(* IEC 61131-3 sources: SJ_AGV/PLC/Vehicle_specfic_functions, 3 files *)

(* ---- BMS_CHG_FB.ST ---- *)
FUNCTION_BLOCK BMS_CHG_FB
VAR_EXTERNAL

END_VAR

VAR_INPUT

END_VAR

VAR_OUTPUT

END_VAR

VAR
	StepDelay : TON;
	ManualStepDelay : TON;
	CheckChargeDoneStepDelay : TON;

	 ChageTimer : TON;
	 ChargeFullFlag : BOOL;

	 AutoChargeStep : INT := 0;
	 ChargePnt : DINT := 0;

	 FastChargeFlag : BOOL;
	 FastChargeTimer : TON;
	 FastChargeTimeOver : BOOL;

END_VAR
(* Check Manual Charge *)

if PLC_RX03_Bit_ChrgReqL_A = TRUE and PLC_TX01_Bit_ManMode = TRUE and PLC_RX03_Bit_Charging_L = FALSE then
	NDC8.SDIO.DigitalOutput16_Charger := TRUE;
	PLC_TX01_Bit_ChrgSelL_A := TRUE;
	StopCharge := TRUE;

	(* Full Charge Point check *)
	if NDC8.PointTrigger.Bit14_Full_Chrg = FALSE then
		PLC_TX01_Bit_TRChg_Pnt := TRUE;
	else
		PLC_TX01_Bit_TRChg_Pnt := FALSE;
	end_if;

	g_BattLim_NG := FALSE;
	INPUT.LowBattery := FALSE;
	NDC8.Userdefined.LowBatSim := FALSE;
	OM_PLC_W1_Bit_SetLowBatt := FALSE;

	ManualStepDelay(IN := TRUE, PT := t#1s);

	if ManualStepDelay.Q Then
		PLC_TX04_Bit_ChrgCmdL_A := TRUE;
		ManualStepDelay(IN := FALSE);
	end_if;

elsif PLC_RX03_Bit_ChrgReqR_A = TRUE and PLC_TX01_Bit_ManMode = TRUE and PLC_RX03_Bit_Charging_R = FALSE then
	NDC8.SDIO.DigitalOutput16_Charger := TRUE;
	PLC_TX01_Bit_ChrgSelR_A := TRUE;
	StopCharge := TRUE;

	(* Full Charge Point check *)
	if NDC8.PointTrigger.Bit14_Full_Chrg = FALSE then
		PLC_TX01_Bit_TRChg_Pnt := TRUE;
	else
		PLC_TX01_Bit_TRChg_Pnt := FALSE;
	end_if;

	g_BattLim_NG := FALSE;
	INPUT.LowBattery := FALSE;
	NDC8.Userdefined.LowBatSim := FALSE;
	OM_PLC_W1_Bit_SetLowBatt := FALSE;

	ManualStepDelay(IN := TRUE, PT := t#1s);

	if ManualStepDelay.Q Then
		PLC_TX04_Bit_ChrgCmdR_A := TRUE;
		ManualStepDelay(IN := FALSE);
	end_if;

elsif (PLC_RX03_Bit_ChrgReqL_A = FALSE and PLC_RX03_Bit_ChrgReqR_A = FALSE) and PLC_TX01_Bit_ManMode = TRUE then
	NDC8.SDIO.DigitalOutput16_Charger := FALSE;

	PLC_TX04_Bit_ChrgCmdL_A := FALSE;
	PLC_TX04_Bit_ChrgCmdR_A := FALSE;

	PLC_TX01_Bit_TRChg_Pnt := FALSE;

	ManualStepDelay(IN := TRUE, PT := t#1s);

	if ManualStepDelay.Q Then
		PLC_TX01_Bit_ChrgSelL_A := FALSE;
		PLC_TX01_Bit_ChrgSelR_A := FALSE;
		StopCharge := FALSE;
		ManualStepDelay(IN := FALSE);
		INPUT.LowBattery := FALSE;
	end_if;

end_if;

case AutoChargeStep of

	0:

		if (INPUT.Auto = TRUE and NDC8.Automatic.ExecDriveCommand = FALSE ) and
			((NDC8.PointTrigger.Bit9_Chrg_Right = TRUE and NDC8.PointTrigger.Bit10_Chrg_Left = FALSE) or (NDC8.PointTrigger.Bit9_Chrg_Right = FALSE and NDC8.PointTrigger.Bit10_Chrg_Left = TRUE)) and
			(PLC_RX01_Bit_ChrgEmg = FALSE) then
			AutoChargeStep := 70;
			g_ChargeDone := FALSE;
			ChargePnt := NDC8.LayoutPosition.Point;
		end_if;

		OM_PLC_Word9 := INT_TO_WORD(NDC8.OMPLC.Round_om);

		OM_PLC_W9_Bit_ChgP_Err := FALSE;

		NDC8.OMPLC.Round_om := WORD_TO_INT(OM_PLC_Word9);

(* Charge the battery Host Order *)
	70:

		if NDC8.PointTrigger.Bit9_Chrg_Right = TRUE and NDC8.PointTrigger.Bit10_Chrg_Left = FALSE then
			PLC_TX01_Bit_ChrgSelR_A := TRUE;
		elsif NDC8.PointTrigger.Bit9_Chrg_Right = FALSE and NDC8.PointTrigger.Bit10_Chrg_Left = TRUE then
			PLC_TX01_Bit_ChrgSelL_A := TRUE;
		end_if;

		(* Full Charge Point check *)
		if NDC8.PointTrigger.Bit14_Full_Chrg = FALSE then
			PLC_TX01_Bit_TRChg_Pnt := TRUE;
		else
			PLC_TX01_Bit_TRChg_Pnt := FALSE;
		end_if;

		OM_PLC_Word9 := INT_TO_WORD(NDC8.OMPLC.Round_om);

		PLC_TX01_Bit_Cancel_ST2 := not OM_PLC_W9_Bit_Enable_Err;
		OM_PLC_W9_Bit_ChgP_Err := FALSE;

		if NDC8.PLC_Application.TxStatusBit9_EStop = TRUE then
			AutoChargeStep := 999;
		elsif PLC_RX01_Bit_ChrgEmg = TRUE then
			AutoChargeStep := 999;
		elsif PLC_RX03_Bit_Round_ChgP = TRUE then
			OM_PLC_W9_Bit_ChgP_Err := TRUE;
			AutoChargeStep := 72;
		elsif PLC_RX01_Bit_ChrgBrk = TRUE then
			AutoChargeStep := 72;
		elsif INPUT.Auto = FALSE then
			AutoChargeStep := 72;
		end_if;

		NDC8.OMPLC.Round_om := WORD_TO_INT(OM_PLC_Word9);

		StopCharge := TRUE;

		(* Check Charge Idle*)
		if PLC_RX03_Bit_CP_HP = TRUE then
			StepDelay(IN:=TRUE, PT:=t#2s);
			if StepDelay.Q then
				StepDelay(IN:=FALSE);
				AutoChargeStep := 71;
			end_if;

		end_if;

	71:

		OM_PLC_Word9 := INT_TO_WORD(NDC8.OMPLC.Round_om);

		PLC_TX01_Bit_Cancel_ST2 := not OM_PLC_W9_Bit_Enable_Err;

		OM_PLC_W9_Bit_ChgP_Err := FALSE;

		if NDC8.PLC_Application.TxStatusBit9_EStop = TRUE then
			AutoChargeStep := 999;
		elsif PLC_RX01_Bit_ChrgEmg = TRUE then
			AutoChargeStep := 999;
		elsif PLC_RX03_Bit_Round_ChgP = TRUE then
			OM_PLC_W9_Bit_ChgP_Err := TRUE;
			AutoChargeStep := 72;
		elsif PLC_RX01_Bit_ChrgBrk = TRUE then
			AutoChargeStep := 72;
		elsif INPUT.Auto = FALSE then
			AutoChargeStep := 72;
		end_if;

		NDC8.OMPLC.Round_om := WORD_TO_INT(OM_PLC_Word9);

		PLC_TX04_Bit_ChrgCmdL_A := NDC8.PointTrigger.Bit10_Chrg_Left;
		PLC_TX04_Bit_ChrgCmdR_A := NDC8.PointTrigger.Bit9_Chrg_Right;

		NDC8.SDIO.DigitalOutput16_Charger := TRUE;

		OM_PLC_Word1 := INT_TO_WORD(NDC8.OMPLC.ChargeOM);
		OM_PLC_Word2 := INT_TO_WORD(NDC8.OMPLC.Stop_OM);

		g_BattLim_NG := FALSE;
		INPUT.LowBattery := FALSE;
		NDC8.Userdefined.LowBatSim := FALSE;
		OM_PLC_W1_Bit_SetLowBatt := FALSE;

		if NDC8.PointTrigger.Bit14_Full_Chrg = TRUE then
			if (g_ChargeDone or PLC_RX01_Bit_ChrgEmg) then
				AutoChargeStep := 72;
			end_if;
		else
			if (NDC8.Automatic.ExecDriveCommand = TRUE or PLC_RX01_Bit_ChrgEmg) or g_ChargeDone or FastChargeTimeOver then
				AutoChargeStep := 72;
			end_if;
		end_if;

	72:

		OM_PLC_Word9 := INT_TO_WORD(NDC8.OMPLC.Round_om);

		PLC_TX01_Bit_Cancel_ST2 := not OM_PLC_W9_Bit_Enable_Err;

		NDC8.OMPLC.Round_om := WORD_TO_INT(OM_PLC_Word9);

		if PLC_RX01_Bit_ChrgEmg = TRUE then
			AutoChargeStep := 999;
		end_if;

		if NDC8.PLC_Application.TxStatusBit9_EStop = TRUE then
			AutoChargeStep := 999;
		end_if;

		PLC_TX04_Bit_ChrgCmdL_A := FALSE;
		PLC_TX04_Bit_ChrgCmdR_A := FALSE;

		NDC8.SDIO.DigitalOutput16_Charger := FALSE;

		OM_PLC_Word1 := INT_TO_WORD(NDC8.OMPLC.ChargeOM);

		OM_PLC_W1_Bit_SetLowBatt := FALSE;

		NDC8.OMPLC.ChargeOM := WORD_TO_INT(OM_PLC_Word1);

		StepDelay(IN:=TRUE, PT:=t#5s);
		if StepDelay.Q then
			StepDelay(IN:=FALSE);
			AutoChargeStep := 73;
		end_if;

	73:

		PLC_TX01_Bit_ChrgSelL_A := FALSE;
		PLC_TX01_Bit_ChrgSelR_A := FALSE;

		OM_PLC_Word9 := INT_TO_WORD(NDC8.OMPLC.Round_om);

		PLC_TX01_Bit_Cancel_ST2 := not OM_PLC_W9_Bit_Enable_Err;

		NDC8.OMPLC.Round_om := WORD_TO_INT(OM_PLC_Word9);

		if PLC_RX01_Bit_ChrgEmg = TRUE then
			AutoChargeStep := 999;
		end_if;

		if NDC8.PLC_Application.TxStatusBit9_EStop = TRUE then
			AutoChargeStep := 999;
		end_if;

		if PLC_RX03_Bit_CP_HP then
			StepDelay(IN:=TRUE, PT:=t#1s);
			if StepDelay.Q then
				StepDelay(IN:=FALSE);
				StopCharge := FALSE;
				AutoChargeStep := 74;
			end_if;
		end_if;

	74:

		OM_PLC_Word9 := INT_TO_WORD(NDC8.OMPLC.Round_om);

		PLC_TX01_Bit_Cancel_ST2 := not OM_PLC_W9_Bit_Enable_Err;

		NDC8.OMPLC.Round_om := WORD_TO_INT(OM_PLC_Word9);

		if PLC_RX01_Bit_ChrgEmg = TRUE then
			AutoChargeStep := 999;
		end_if;

		if NDC8.PLC_Application.TxStatusBit9_EStop = TRUE then
			AutoChargeStep := 999;
		end_if;

		if INPUT.Auto = FALSE then
			AutoChargeStep := 0;
		end_if;

		if NDC8.LayoutPosition.Point <> ChargePnt or NDC8.PLC_Application.TxStatusBit4_LowBatt = TRUE then
			AutoChargeStep := 0;
		end_if;

	999:
		PLC_TX04_Bit_ChrgCmdL_A := FALSE;
		PLC_TX04_Bit_ChrgCmdR_A := FALSE;

		PLC_TX01_Bit_TRChg_Pnt := FALSE;

		StepDelay(IN:=TRUE, PT:=t#1s);
		if StepDelay.Q then
			StepDelay(IN:=FALSE);
			PLC_TX01_Bit_ChrgSelL_A := FALSE;
			PLC_TX01_Bit_ChrgSelR_A := FALSE;
			AutoChargeStep := 0;
			INPUT.LowBattery := FALSE;
		end_if;

		NDC8.SDIO.DigitalOutput16_Charger := FALSE;

		OM_PLC_Word1 := INT_TO_WORD(NDC8.OMPLC.ChargeOM);

		OM_PLC_W1_Bit_SetLowBatt := FALSE;

		NDC8.OMPLC.ChargeOM := WORD_TO_INT(OM_PLC_Word1);

		StopCharge := FALSE;

end_case;

(* Charge Complete Check *)
if (NDC8.PointTrigger.Bit9_Chrg_Right = TRUE or NDC8.PointTrigger.Bit10_Chrg_Left = TRUE) or PLC_TX01_Bit_ManMode = TRUE then
	if(NDC8.CAN_IO_3.DigitalInput5_BatTmp25_i = TRUE and
		NDC8.CAN_IO_3.DigitalInput6_BatTmp40_i = TRUE and
		NDC8.CAN_IO_3.DigitalInput7_BatTmp55_i = TRUE and
		g_BatteryVoltage >= NDC8.UserDefined.Integer32_40_ChgComV1) then
		g_ChargeDone := TRUE;
		g_ChargeTempErr := FALSE;
	elsif (NDC8.CAN_IO_3.DigitalInput5_BatTmp25_i = FALSE and
		NDC8.CAN_IO_3.DigitalInput6_BatTmp40_i = TRUE and
		NDC8.CAN_IO_3.DigitalInput7_BatTmp55_i = TRUE and
		g_BatteryVoltage >= NDC8.UserDefined.Integer32_41_ChgComV2) then
		g_ChargeDone := TRUE;
		g_ChargeTempErr := FALSE;
	elsif (NDC8.CAN_IO_3.DigitalInput5_BatTmp25_i = FALSE and
		NDC8.CAN_IO_3.DigitalInput6_BatTmp40_i = FALSE and
		NDC8.CAN_IO_3.DigitalInput7_BatTmp55_i = TRUE and
		g_BatteryVoltage >= NDC8.UserDefined.Integer32_42_ChgComV3) then
		g_ChargeDone := TRUE;
		g_ChargeTempErr := FALSE;
	elsif (NDC8.CAN_IO_3.DigitalInput5_BatTmp25_i = FALSE and
		NDC8.CAN_IO_3.DigitalInput6_BatTmp40_i = FALSE and
		NDC8.CAN_IO_3.DigitalInput7_BatTmp55_i = FALSE) then
		g_ChargeDone := FALSE;
		g_ChargeTempErr := TRUE;
	else
		g_ChargeDone := FALSE;
		g_ChargeTempErr := FALSE;
	end_if;

elsif (NDC8.CAN_IO_3.DigitalInput5_BatTmp25_i = FALSE and
		NDC8.CAN_IO_3.DigitalInput6_BatTmp40_i = FALSE and
		NDC8.CAN_IO_3.DigitalInput7_BatTmp55_i = FALSE) then

	g_ChargeDone := FALSE;
	g_ChargeTempErr := TRUE;
else
	g_ChargeDone := FALSE;
	g_ChargeTempErr := FALSE;
end_if;

(* Charge Over Time Check *)

	ChargeFullFlag  := NDC8.SDIO.DigitalOutput16_Charger = TRUE and NDC8.PointTrigger.Bit14_Full_Chrg = TRUE;

	ChageTimer(IN:= ChargeFullFlag, PT:=t#1800s);

	if ChageTimer.Q then
		g_ChargeOverTime := TRUE;
	end_if;

	if ChargeFullFlag = FALSE then
		g_ChargeOverTime := FALSE;
	end_if;

(* Fast Charge Time Check *)

	FastChargeFlag := NDC8.SDIO.DigitalOutput16_Charger = TRUE and NDC8.PointTrigger.Bit14_Full_Chrg = FALSE;

	FastChargeTimer(IN:= FastChargeFlag, PT:=t#600s);

	if FastChargeTimer.Q then
		FastChargeTimeOver := TRUE;
	end_if;

	if FastChargeFlag = FALSE then
		FastChargeTimeOver := FALSE;
	end_if;

(* Check BMS Error Status *)
if NDC8.SDIO.DigitalInput2_BTN_RST = FALSE and
	(PLC_RX01_Bit_ChrgEmg = TRUE
	or g_ChargeDone = TRUE
	or g_ChargeOverTime = TRUE
	or g_ChargeTempErr = TRUE) then

		PLC_TX04_Bit_ChrgCmdL_A := FALSE;
		PLC_TX04_Bit_ChrgCmdR_A := FALSE;

		NDC8.SDIO.DigitalOutput16_Charger := FALSE;

		CheckChargeDoneStepDelay(IN := TRUE, PT := t#1s);

		if CheckChargeDoneStepDelay.Q then
			CheckChargeDoneStepDelay(IN := FALSE);
			PLC_TX01_Bit_ChrgSelL_A := FALSE;
			PLC_TX01_Bit_ChrgSelR_A := FALSE;
		end_if;

end_if;

(* Let Vehicle Stop *)
(*
if PLC_TX04_Bit_ChrgCmdL_A = TRUE or PLC_TX04_Bit_ChrgCmdR_A = TRUE or
	PLC_RX03_Bit_CP_HP = FALSE or
	AutoChargeStep = 70 or AutoChargeStep = 71 or AutoChargeStep = 72 or AutoChargeStep = 73 then
	StopCharge := TRUE;
end_if;
*)

END_FUNCTION_BLOCK

(* ---- MITSUBISHIMODBUS_FB.ST ---- *)
FUNCTION_BLOCK MITSUBISHIMODBUS_FB
VAR_EXTERNAL

	ConvWord:WORD;			(*Sum of the two first bytes*)

	ConvByteL:Byte;			(*Low byte*)
	ConvByteH:Byte;			(*High byte*)
END_VAR

VAR_INPUT
	ComStart : bool := TRUE;
END_VAR

VAR_OUTPUT

END_VAR

VAR
	BMS_BatLowSel : INT;
	BMS_BatLow : BOOL;

	TP_PB_NoSelTimer : TON;

	Debug_PB_Cont : BOOL := FALSE;
	Debug_PB_Finish : BOOL := FALSE;
	Debug_PB_Cancel : BOOL := FALSE;
	Debug_PB_Change : BOOL := FALSE;

	RST_Flag : BOOL;
	RST_R : R_Trig;

	RST_Keep : BOOL;
	RST_Keep_Timer : TON;

	BatLow : BOOL;

	TempInt : int;
	TempWord : word;
	WordL :int;
	WordH :int;

	FinalPnt : DINT;

	SwitchHostFlag : BOOL;
	Host_R : R_Trig;
	Host_R_Flag : BOOL;

	Host_R_Delay : TON;

	init  : bool := false;
	ComStep : int := 0;

	serial_read : NDC8_SERIAL_READ;
	serial_write : NDC8_SERIAL_WRITE;

	to_bytes 		: NDC8_STRING_TO_BYTES;
	to_string		: NDC8_BYTES_TO_STRING;

	PLC_LastHeartBeat : BOOL;
	PLC_HeartBeatNoChange : BOOL;

	PLC_HeartBeatTimeout : TON;

	LoadDataSendFlag : BOOL;
	UnloadDataSendFlag : BOOL;

	TestDataSend : BOOL;

	OrderMode:OrderMode_FB;
	LocalOrder : LocalOrder_FB;
	NavInit : NavInit_FB;

	STw_NewcmdR : R_Trig;
	STw_Newcmd_Flag : BOOL;

	LocalManual : BOOL;
	LocalManual_R : R_Trig;
	SetToLocal : BOOL;

	Str_AckT : TON;
	STr_AckR : BOOL;

	(*---------Rev Data ----------*)
	Start : int;
	StartOffset : int;

	DataIndex1 : Int;
	DataIndex2 : Int;
	DataIndex3 : Int;
	DataIndex4 : Int;
	DataIndex5 : Int;

	RevDataLength : int := 0;

	TempString : string;

	HeaderString : string;
	DecodeString : string(200);
	DecodeString_RS : string(200);
	DecodeString_WS : string(200);

	TempData : ARRAY[1..32] OF BYTE;

	SendData_Req : ARRAY[1..32] OF BYTE;

	ReceiveData_Status : ARRAY[1..1074] OF BYTE;
	(*--------------------------------------*)

	(*Send 16 Word Data *)
	EncoderStart : int;
	EncoderStartOffset : int;
	MessageLen : int;

	Message : string;
	SendTempString : string;

	SendData_Status1 : ARRAY[1..32] OF BYTE;
	SendData_Status2 : ARRAY[1..32] OF BYTE;
	SendData_Status3 : ARRAY[1..32] OF BYTE;
	SendData_Status4 : ARRAY[1..32] OF BYTE;

	(*--------------------------------------*)

	(*Decode WS Data*)
	DecodeStart_WS : int;

	DecodeString_WS_Data :string(200);
	SplitString : string;

	SplitPos : int;
	SplitPosOffset1 : int;

	DecodeDataArray : ARRAY[1..25] of WORD;

	(*---------------------------------------*)
	tx_header_length : BYTE := 6;
	dummy : BOOL;
	tr_cmd : DINT;

	start_adress : INT;

	ReadCounter,
	DebugCounter		: DINT;
	StartDelayTOF	: TOF;
	StartDelay 		: BOOL;

	X: INT;
	Y: INT;
	Z: INT;
	End:INT;
	Index:DINT;
	debug1 :INT;
	debug2 :INT;
	tr_len : DINT;
	num_words : DINT;
	num_Byte : DINT;
	num_Bit : DINT;
	Extra:DINT;
	length : DINT;
	tx_length : BYTE;
	ENDBIT:DINT;
	debugByte :Byte;
	dataindex : INT;
	msg_index: INT;
	ix : INT;
	PLC_message : ARRAY[1..500] of BYTE;
	lenght_send : DINT;
	Send_message : ARRAY[1..32] of BYTE;
	Counter : DINT;
	DINTdataindex : DINT;
	WRITENUM : INT;

END_VAR
StartDelayTOF(IN:=StartDelay, PT:=t#20ms);
if init = false then
	serial_read.port := 'COM7';
	serial_write.port := 'COM7';
	init := true;
end_if;

(*Communication*)

(****************************************************************************)
if ComStart = true then

	if init = true then
		case ComStep of
		0:
		StartDelay:=False;
		IF NOT StartDelayTOF.Q THEN
			ComStep:=1;
		END_IF;
		(* no delay when PLC <--> CVC700*)
		(****************************************************************************)
		1:
			msg_index := 0;
			serial_read();

			while serial_read.length > 0 do
					(* Copy message to local buffer *)
					for dataindex := 1 to serial_read.length by 1 do
						ix := dataindex + msg_index;
						PLC_message[ix] := serial_read.data[dataindex];
					end_for;
					(* Point for next possible message *)
					msg_index := msg_index + serial_read.length;
				end_if;
				serial_read();
			end_while;
			if msg_index <> 0 then
				ComStep:=2;
			END_IF;
			if msg_index = 0 then
				ComStep:=0;
			END_IF;

		(****************************************************************************)
		2:
				    (* Parse *)
					tr_cmd := BYTE_TO_DINT(PLC_message[8]);
					tr_len := BYTE_TO_DINT(PLC_message[6]);

					dummy := TRACE_DINT('Cmd', tr_cmd);
					dummy := TRACE_DINT('Len', tr_len);

					(* Copy header *)
					serial_write.data[1] := PLC_message[1];
					serial_write.data[2] := PLC_message[2];
					serial_write.data[3] := PLC_message[3];
					serial_write.data[4] := PLC_message[4];
					serial_write.data[5] := PLC_message[5];		(* Length, will be overwritten *)

					serial_write.data[6] := PLC_message[6]; 	(* Length, will be overwritten *)
					serial_write.data[7] := PLC_message[7]; 	(* Slave adress *)
					serial_write.data[8] := PLC_message[8]; 	(* Cmd *)

					(* Start adress to read *)
					ConvByteH:= PLC_message[9];
					ConvByteL:= PLC_message[10];
					start_adress  := Word_TO_INT(ConvWord) + 1;

					ComStep:=3;

					(*if STOPNUM <> 0 then
						ComStep:=2;
						STOPVAL := PLC_message[STOPINX];
					end_if;*)
		(****************************************************************************)
		3:

					(*Check Function type *)
				    STOPNUM := DINT_TO_INT(tr_cmd);
					case tr_cmd of
						6:	ComStep:=160;	(* Check if Write single register *)
						16:	ComStep:=160; (* Check if write Multiple register *)
						10: ComStep:=160;
						3:	ComStep:=30;	(*Check if Read register *)
					Else
						ComStep:=0; 	(*Send Echo *)
					end_case;
		(****************************************************************************)
		30:
						(*Read register *)
						(* Number of words *)
						(* serial_read.data[11]; *)
						(*CVC700 -> PLC HandShake Data*)
						PLC_Communication_ModBus_ValueWord [1] := PLC_TX_Word1;
						PLC_Communication_ModBus_ValueWord [2] := PLC_TX_Word2;
						PLC_Communication_ModBus_ValueWord [3] := PLC_TX_Word3;
						PLC_Communication_ModBus_ValueWord [4] := PLC_TX_Word4;
						PLC_Communication_ModBus_ValueWord [5] := PLC_TX_Word5;
						PLC_Communication_ModBus_ValueWord [6] := PLC_TX_Word6;
						PLC_Communication_ModBus_ValueWord [7] := PLC_TX_Word7_STr_Vecl;
						PLC_Communication_ModBus_ValueWord [8] := PLC_TX_Word8_STr_Seg;
						PLC_Communication_ModBus_ValueWord [9] := PLC_TX_Word9_STr_Pnt;
						PLC_Communication_ModBus_ValueWord [10] := PLC_TX_Word10_STr_BatV;
						PLC_Communication_ModBus_ValueWord [11] := PLC_TX_Word11_STr_Temp;
						PLC_Communication_ModBus_ValueWord [12] := PLC_TX_Word12_STr_BatD;
						PLC_Communication_ModBus_ValueWord [13] := PLC_TX_Word13_STr_Err;
						PLC_Communication_ModBus_ValueWord [14] := PLC_TX_Word14_STr_BCD3;
						PLC_Communication_ModBus_ValueWord [15] := PLC_TX_Word15_STr_BCD2;
						PLC_Communication_ModBus_ValueWord [16] := PLC_TX_Word16_STr_BCD1;
						num_words := BYTE_TO_DINT(PLC_message[12]);

						(*IF num_words >21 THEN
						   	num_words:=21;
						END_IF;*)

							(*Y:=start_adress;*)
							Y := start_adress;
							(* Copy header *)
							serial_write.data[1] := PLC_message[1];
							serial_write.data[2] := PLC_message[2];
							serial_write.data[3] := PLC_message[3];
							serial_write.data[4] := PLC_message[4];
							serial_write.data[5] := PLC_message[5];
							Z:= 1; (* Send first 9*)
							serial_write.data[6] := DINT_TO_BYTE(35); (* lp *)
							serial_write.data[7] := PLC_message[7]; 	(* Slave adress *)
							serial_write.data[8] := PLC_message[8]; 	(* Cmd *)
							serial_write.data[9] := DINT_TO_BYTE(32); (* lp *)
				        	serial_write.length := 9;
							serial_write();
							serial_write.length := 0; (*Using SendBuffer =1 length needs to be set to 0 for it to be sent*)
							serial_write(); (*send*)
							While Total > 0 Then
								Total := Total - 16;
								IF Total > 0 THEN
									For Index:=1 to 16 BY 1 DO
										ConvWord:=PLC_Communication_ModBus_ValueWord [Y];
										serial_write.data[Z]:=ConvByteH;
										Z:=Z+1;
										serial_write.data[Z]:=ConvByteL;
										Z:=Z+1;
										Y:=Y+1;
									END_FOR;
									serial_write.length := DINT_TO_INT(16); (*Will be max 32 bytes*)
									serial_write();
									serial_write.length := 0; (*Using SendBuffer =1 length needs to be set to 0 for it to be sent*)
									serial_write(); (*send*)
								ESLE
									For Index:=1 to (TOTAL + 16) BY 1 DO
										ConvWord:=PLC_Communication_ModBus_ValueWord [Y];
										serial_write.data[Z]:=ConvByteH;
										Z:=Z+1;
										serial_write.data[Z]:=ConvByteL;
										Z:=Z+1;
										Y:=Y+1;
									END_FOR;
									serial_write.length := DINT_TO_INT(TOTAL + 16); (*Will be max 32 bytes*)
									serial_write();
									serial_write.length := 0; (*Using SendBuffer =1 length needs to be set to 0 for it to be sent*)
									serial_write(); (*send*)
								END_IF;
							End_If;
							ComStep:=10001;

		(****************************************************************************)
		160:

						(* Multiple write *)
						num_words:=Byte_TO_DInt(PLC_message[12]);
						(* Check if message lenght outside the Buffer, if so do what ??? *)
						Y:=start_adress;
						X:=14;  (*13 = How many bytes will send after 13 this byte)
						End:= Byte_TO_Int(PLC_message[12]);

						For Index:=1 to num_words BY 1 DO
							ConvByteH:=PLC_message[X];
							X:=X+1;
							ConvByteL:=PLC_message[X];
							PLC_Communication_ModBus_ValueWord [Y]:=ConvWord;
							X:=X+1;
							Y:=Y+1;
						END_FOR;
						(*Set Into Memory *)
						PLC_RX_Word1 := PLC_Communication_ModBus_ValueWord [17];
						PLC_RX_Word2 := PLC_Communication_ModBus_ValueWord [18];
						PLC_RX_Word3 := PLC_Communication_ModBus_ValueWord [19];
						PLC_RX_Word4 := PLC_Communication_ModBus_ValueWord [20];
						PLC_RX_Word5 := PLC_Communication_ModBus_ValueWord [21];
						PLC_RX_Word6 := PLC_Communication_ModBus_ValueWord [22];
						PLC_RX_Word7_STw_BCD3 := PLC_Communication_ModBus_ValueWord [23];
						PLC_RX_Word8_STw_BCD2 := PLC_Communication_ModBus_ValueWord [24];
						PLC_RX_Word9_STw_BCD1 := PLC_Communication_ModBus_ValueWord [25];
						PLC_RX_Word10_STw_ILEr := PLC_Communication_ModBus_ValueWord [26];
						PLC_RX_Word11_Ins_Pno := PLC_Communication_ModBus_ValueWord [27];
						PLC_RX_Word12_STw_Pint := PLC_Communication_ModBus_ValueWord [28];
						PLC_RX_Word13_Ins_Ano := PLC_Communication_ModBus_ValueWord [29];
						PLC_RX_Word14_BMS_2 := PLC_Communication_ModBus_ValueWord [30];
						PLC_RX_Word15_BMS_3 := PLC_Communication_ModBus_ValueWord [31];
						PLC_RX_Word16_BMS_BatV := PLC_Communication_ModBus_ValueWord [32];
						PLC_RX_Word17_BMS_BatT := PLC_Communication_ModBus_ValueWord [33];
						PLC_RX_Word18_BMS_BatC := PLC_Communication_ModBus_ValueWord [34];
						PLC_RX_Word19_BMS_BatA := PLC_Communication_ModBus_ValueWord [35];
						PLC_RX_Word20_PLC_ErrD := PLC_Communication_ModBus_ValueWord [36];
						PLC_RX_Word21_BMS_Main := PLC_Communication_ModBus_ValueWord [37];
						PLC_RX_Word22_BMS_Chan := PLC_Communication_ModBus_ValueWord [38];
						PLC_RX_Word23_BMS_ID4L := PLC_Communication_ModBus_ValueWord [39];
						PLC_RX_Word24_BMS_ID4H := PLC_Communication_ModBus_ValueWord [40];
						PLC_RX_Word25 := PLC_Communication_ModBus_ValueWord [41];
						ComStep := 999;
		(****************************************************************************)
		999:
					Serial_write.data[1] := PLC_message[1];
					Serial_write.data[2] := PLC_message[2];
					Serial_write.data[3] := PLC_message[3];
					Serial_write.data[4] := PLC_message[4];
					Serial_write.data[5] := PLC_message[5];
				    Serial_write.data[6] := DINT_TO_BYTE(57);
					Serial_write.data[7] := PLC_message[7];
					Serial_write.data[8] := PLC_message[8];
					Serial_write.data[9] := PLC_message[9];
					serial_write.data[10] := PLC_message[10];
					serial_write.data[11] := PLC_message[11];
					serial_write.data[12] := DINT_TO_BYTE(25);   (*PLC_message[12];*)
					serial_write.length := 12;
					serial_write();
					PLC_message[8] := 0;
					ComStep:=10001;
					WRITENUM := WRITENUM + 1;
		(****************************************************************************)
		10000:

					(*Send Data *)

					serial_write.length := 0;
					serial_write();
					IF serial_write.sent<>0 or serial_write.error<>0 Then
						ComStep:=0;
						DebugCounter := DebugCounter + 1;
					End_IF;
					ComStep:=0;
		10001:
					serial_write.length := 0; (*Using SendBuffer =1 length needs to be set to 0 for it to be sent*)
					serial_write(); (*send*)
					IF serial_write.sent<>0 or serial_write.error<>0 Then
						ComStep:=0;
						DebugCounter := DebugCounter + 1;
					End_IF;
					ComStep:=0;
		end_case;

	(*CVC700 -> PLC HandShake Data*)
	(*PLC_Communication_ModBus_ValueWord [1] := PLC_TX_Word1;
	PLC_Communication_ModBus_ValueWord [2] := PLC_TX_Word2;
	PLC_Communication_ModBus_ValueWord [3] := PLC_TX_Word3;
	PLC_Communication_ModBus_ValueWord [4] := PLC_TX_Word4;
	PLC_Communication_ModBus_ValueWord [5] := PLC_TX_Word5;
	PLC_Communication_ModBus_ValueWord [6] := PLC_TX_Word6;
	PLC_Communication_ModBus_ValueWord [7] := PLC_TX_Word7_STr_Vecl;
	PLC_Communication_ModBus_ValueWord [8] := PLC_TX_Word8_STr_Seg;
	PLC_Communication_ModBus_ValueWord [9] := PLC_TX_Word9_STr_Pnt;
	PLC_Communication_ModBus_ValueWord [10] := PLC_TX_Word10_STr_BatV;
	PLC_Communication_ModBus_ValueWord [11] := PLC_TX_Word11_STr_Temp;
	PLC_Communication_ModBus_ValueWord [12] := PLC_TX_Word12_STr_BatD;
	PLC_Communication_ModBus_ValueWord [13] := PLC_TX_Word13_STr_Err;
	PLC_Communication_ModBus_ValueWord [14] := PLC_TX_Word14_STr_BCD3;
	PLC_Communication_ModBus_ValueWord [15] := PLC_TX_Word15_STr_BCD2;
	PLC_Communication_ModBus_ValueWord [16] := PLC_TX_Word16_STr_BCD1;
	*)

	(*PLC -> CVC700 HandShake Data*)
	(*PLC_RX_Word1 := PLC_Communication_ModBus_ValueWord [17];
	PLC_RX_Word2 := PLC_Communication_ModBus_ValueWord [18];
	PLC_RX_Word3 := PLC_Communication_ModBus_ValueWord [19];
	PLC_RX_Word4 := PLC_Communication_ModBus_ValueWord [20];
	PLC_RX_Word5 := PLC_Communication_ModBus_ValueWord [21];
	PLC_RX_Word6 := PLC_Communication_ModBus_ValueWord [22];
	PLC_RX_Word7_STw_BCD3 := PLC_Communication_ModBus_ValueWord [23];
	PLC_RX_Word8_STw_BCD2 := PLC_Communication_ModBus_ValueWord [24];
	PLC_RX_Word9_STw_BCD1 := PLC_Communication_ModBus_ValueWord [25];
	PLC_RX_Word10_STw_ILEr := PLC_Communication_ModBus_ValueWord [26];
	PLC_RX_Word11_Ins_Pno := PLC_Communication_ModBus_ValueWord [27];
	PLC_RX_Word12_STw_Pint := PLC_Communication_ModBus_ValueWord [28];
	PLC_RX_Word13_Ins_Ano := PLC_Communication_ModBus_ValueWord [29];
	PLC_RX_Word14_BMS_2 := PLC_Communication_ModBus_ValueWord [30];
	PLC_RX_Word15_BMS_3 := PLC_Communication_ModBus_ValueWord [31];
	PLC_RX_Word16_BMS_BatV := PLC_Communication_ModBus_ValueWord [32];
	PLC_RX_Word17_BMS_BatT := PLC_Communication_ModBus_ValueWord [33];
	PLC_RX_Word18_BMS_BatC := PLC_Communication_ModBus_ValueWord [34];
	PLC_RX_Word19_BMS_BatA := PLC_Communication_ModBus_ValueWord [35];
	PLC_RX_Word20_PLC_ErrD := PLC_Communication_ModBus_ValueWord [36];
	PLC_RX_Word21_BMS_Main := PLC_Communication_ModBus_ValueWord [37];
	PLC_RX_Word22_BMS_Chan := PLC_Communication_ModBus_ValueWord [38];
	PLC_RX_Word23_BMS_ID4L := PLC_Communication_ModBus_ValueWord [39];
	PLC_RX_Word24_BMS_ID4H := PLC_Communication_ModBus_ValueWord [40];
	PLC_RX_Word25 := PLC_Communication_ModBus_ValueWord [41];
	*)
	end_if;

end_if;

END_FUNCTION_BLOCK

(* ---- PLC_COMMUNICATION_FB.ST ---- *)
FUNCTION_BLOCK PLC_COMMUNICATION_FB
VAR_EXTERNAL

pConvWord:WORD;			(*Sum of the two first bytes*)

pConvByteL:Byte;			(*Low byte*)
pConvByteH:Byte;			(*High byte*)
END_VAR

VAR_INPUT
	ComStart : bool := TRUE;
END_VAR

VAR_OUTPUT

END_VAR

VAR
	BMS_BatLowSel : INT;
	BMS_BatLow : BOOL;

	TP_PB_NoSelTimer : TON;

	Debug_PB_Cont : BOOL := FALSE;
	Debug_PB_Finish : BOOL := FALSE;
	Debug_PB_Cancel : BOOL := FALSE;
	Debug_PB_Change : BOOL := FALSE;

	RST_Flag : BOOL;
	RST_R : R_Trig;

	RST_Keep : BOOL;
	RST_Keep_Timer : TON;

	BatLow : BOOL;

	TempInt : int;
	TempWord : word;
	WordL :int;
	WordH :int;

	FinalPnt : DINT;

	SwitchHostFlag : BOOL;
	Host_R : R_Trig;
	Host_R_Flag : BOOL;

	Host_R_Delay : TON;

	init  : bool := false;
	ComStep : int := 0;

	serial_read : NDC8_SERIAL_READ;
	serial_write : NDC8_SERIAL_WRITE;

	to_bytes 		: NDC8_STRING_TO_BYTES;
	to_string		: NDC8_BYTES_TO_STRING;

	PLC_LastHeartBeat : BOOL;
	PLC_HeartBeatNoChange : BOOL;

	PLC_HeartBeatTimeout : TON;

	LoadDataSendFlag : BOOL;
	UnloadDataSendFlag : BOOL;

	TestDataSend : BOOL;

	OrderMode:OrderMode_FB;
	LocalOrder : LocalOrder_FB;
	NavInit : NavInit_FB;

	STw_NewcmdR : R_Trig;
	STw_Newcmd_Flag : BOOL;

	LocalManual : BOOL;
	LocalManual_R : R_Trig;
	SetToLocal : BOOL;

	Str_AckT : TON;
	STr_AckR : BOOL;

	(*---------Rev Data ----------*)
	Start : int;
	StartOffset : int;

	DataIndex1 : Int;
	DataIndex2 : Int;
	DataIndex3 : Int;
	DataIndex4 : Int;
	DataIndex5 : Int;

	RevDataLength : int := 0;

	TempString : string;

	HeaderString : string;
	DecodeString : string(200);
	DecodeString_RS : string(200);
	DecodeString_WS : string(200);

	TempData : ARRAY[1..32] OF BYTE;

	SendData_Req : ARRAY[1..32] OF BYTE;

	ReceiveData_Status : ARRAY[1..1074] OF BYTE;
	(*--------------------------------------*)

	(*Send 16 Word Data *)
	EncoderStart : int;
	EncoderStartOffset : int;
	MessageLen : int;

	Message : string;
	SendTempString : string;

	SendData_Status1 : ARRAY[1..32] OF BYTE;
	SendData_Status2 : ARRAY[1..32] OF BYTE;
	SendData_Status3 : ARRAY[1..32] OF BYTE;
	SendData_Status4 : ARRAY[1..32] OF BYTE;

	(*--------------------------------------*)

	(*Decode WS Data*)
	DecodeStart_WS : int;

	DecodeString_WS_Data :string(200);
	SplitString : string;

	SplitPos : int;
	SplitPosOffset1 : int;

	DecodeDataArray : ARRAY[1..25] of WORD;

	(*---------------------------------------*)
	tx_header_length : BYTE := 6;
	dummy : BOOL;
	tr_cmd : DINT;

	start_adress : INT;

	ReadCounter,
	DebugCounter		: DINT;
	StartDelayTOF	: TOF;
	StartDelay 		: BOOL;

	X: INT;
	Y: INT;
	Z: INT;
	End:INT;
	Index:DINT;
	debug1 :INT;
	debug2 :INT;
	tr_len : DINT;
	num_words : DINT;
	num_Byte : DINT;
	num_Bit : DINT;
	Extra:DINT;
	length : DINT;
	tx_length : BYTE;
	ENDBIT:DINT;
	debugByte :Byte;
	dataindex : INT;
	msg_index: INT;
	ix : INT;
	PLC_message : ARRAY[1..300] of BYTE;
	lenght_send : DINT;
	Send_message : ARRAY[1..32] of BYTE;
	Counter : DINT;
	DINTdataindex : DINT;
END_VAR
if init = false then
	serial_read.port := 'COM7';
	serial_write.port := 'COM7';
	init := true;
end_if;

(*TX Data Proc*)
(*I00800*)

SwitchHostFlag := INPUT.Auto = TRUE and INPUT.StartMode = TRUE and NDC8.LayoutPosition.InSystem and NDC8.Master.MasterLinkUp;

Host_R(CLK:= SwitchHostFlag);

if SwitchHostFlag then

	Host_R_Delay(IN:= PLC_RX01_Bit_EnableLD_i, PT:=t#1s);

	if Host_R.Q then
		Host_R_Flag := TRUE;
	end_if;

	if NDC8.UserDefined.Boolean_20_OnlineOrderMode = FALSE  then

		if NDC8.Automatic.CurrentOrderMode = 1 then
			Host_R_Flag := FALSE;
		end_if;

		if NDC8.Automatic.CurrentOrderMode <> 1 and Host_R_Flag = TRUE and PLC_RX01_Bit_EnableLD_i = TRUE and Host_R_Delay.Q then
			NDC8.Automatic.SetOrderMode := 1;
			OrderMode();
		elsif NDC8.Automatic.CurrentOrderMode <> 1 and Host_R_Flag = FALSE then
			;
		end_if;
	else
		if NDC8.Automatic.CurrentOrderMode = 3 then
			Host_R_Flag := FALSE;
		end_if;

		if NDC8.Automatic.CurrentOrderMode <> 3 and Host_R_Flag = TRUE and PLC_RX01_Bit_EnableLD_i = TRUE and Host_R_Delay.Q then
			NDC8.Automatic.SetOrderMode := 3;
			OrderMode();
		elsif NDC8.Automatic.CurrentOrderMode <> 3 and Host_R_Flag = FALSE then
			;
		end_if;
	end_if;

else
	PLC_TX01_Bit_HostMode := false;
end_if;

(*I00801*)

PLC_TX01_Bit_ManMode := NDC8.Mcd.Button3;

if PLC_TX01_Bit_ManMode = TRUE then
	INPUT.StartMode := FALSe;
	OM_PLC_Word2 := INT_TO_WORD(NDC8.OMPLC.Stop_OM);
		OM_PLC_W2_Bit_SetEmgStop := FALSE;
	NDC8.OMPLC.Stop_OM := WORD_TO_INT(OM_PLC_Word2);
end_if;

(*I00802*)
if INPUT.Auto = TRUE and (NDC8.Automatic.CurrentOrderMode = 2 or NDC8.Automatic.CurrentOrderMode = 3) then
	PLC_TX01_Bit_HostMode := false;
	PLC_TX01_Bit_LocalMode := true;

elsif INPUT.Auto = TRUE and NDC8.Automatic.CurrentOrderMode = 1 then
	PLC_TX01_Bit_HostMode := true;
	PLC_TX01_Bit_LocalMode := false;
else
	PLC_TX01_Bit_HostMode := false;
	PLC_TX01_Bit_LocalMode := false;
end_if;

(* I00803 *)
if INPUT.StartMode and (PLC_TX01_Bit_HostMode = true or PLC_TX01_Bit_LocalMode = true) and PLC_HeartBeatTimeout.Q = FALSE then
	PLC_TX01_Bit_OnLn_ModeP := TRUE;
else
	PLC_TX01_Bit_OnLn_ModeP := FALSE;
end_if;

if NDC8.Automatic.CurrentOrderMode = 2 then
	PLC_TX01_Bit_STr_Mod_NT := TRUE;
	PLC_TX01_Bit_STr_Mod_UT := FALSE;
elsif NDC8.Automatic.CurrentOrderMode = 1 or NDC8.Automatic.CurrentOrderMode = 3 then
	PLC_TX01_Bit_STr_Mod_NT := FALSE;
	PLC_TX01_Bit_STr_Mod_UT := TRUE;
end_if;

(* I00808 *)

if g_PlcComLinkUp = TRUE then
	if INPUT.LowBattery then
		PLC_TX01_Bit_STr_BatLow := TRUE;
	else
		PLC_TX01_Bit_STr_BatLow := FALSE;
	end_if;
end_if;

(* I00809 *)
	PLC_TX01_Bit_STr_Home := NDC8.PointTrigger.Bit8_HP_Pnt;

(* I00810 *)

STr_AckT(IN := STr_AckR, PT:= t#10s);

if PLC_TX01_Bit_OnLn_ModeP = TRUE then

	if 	PLC_RX04_Bit_STw_Cont = TRUE
		or PLC_RX04_Bit_STw_Finish = TRUE
		or PLC_RX04_Bit_STw_Cancel = TRUE
		or PLC_RX04_Bit_STw_Change = TRUE then

		TP_PB_NoSelTimer(IN:= FALSE);

		OM_PLC_Word1 := INT_TO_WORD(NDC8.OMPLC.ChargeOM);

		OM_PLC_W1_Bit_OM_Cont			:= PLC_RX04_Bit_STw_Cont;
		OM_PLC_W1_Bit_OM_Finish			:= PLC_RX04_Bit_STw_Finish;
		OM_PLC_W1_Bit_OM_Cancel			:= PLC_RX04_Bit_STw_Cancel;
		OM_PLC_W1_Bit_OM_Change			:= PLC_RX04_Bit_STw_Change;

		NDC8.OMPLC.ChargeOM := WORD_TO_INT(OM_PLC_Word1);

		STr_AckR := TRUE;

		if STr_AckT.Q then
			PLC_TX01_Bit_STr_Ack := TRUE;
		else
			PLC_TX01_Bit_STr_Ack := FALSE;
		end_if;

	elsif PLC_RX04_Bit_STw_Cont = FALSE
		or PLC_RX04_Bit_STw_Finish = FALSE
		or PLC_RX04_Bit_STw_Cancel = FALSE
		or PLC_RX04_Bit_STw_Change = FALSE then

		OM_PLC_Word1 := INT_TO_WORD(NDC8.OMPLC.ChargeOM);

		TP_PB_NoSelTimer(IN:=TRUE, PT:= t#10s);

		OM_PLC_W1_Bit_OM_Cont			:= FALSE;
		OM_PLC_W1_Bit_OM_Finish			:= FALSE;
		OM_PLC_W1_Bit_OM_Cancel			:= FALSE;
		OM_PLC_W1_Bit_OM_Change			:= FALSE;

		if TP_PB_NoSelTimer.Q then
			OM_PLC_W1_Bit_OM_Cont := TRUE;
		end_if;

		if Debug_PB_Cont = TRUE then
			OM_PLC_W1_Bit_OM_Cont := TRUE;
		end_if;

		if Debug_PB_Finish = TRUE then
			OM_PLC_W1_Bit_OM_Finish := TRUE;
		end_if;

		if Debug_PB_Cancel = TRUE then
			OM_PLC_W1_Bit_OM_Cancel := TRUE;
		end_if;

		if Debug_PB_Change = TRUE then
			OM_PLC_W1_Bit_OM_Change := TRUE;
		end_if;

		NDC8.OMPLC.ChargeOM := WORD_TO_INT(OM_PLC_Word1);

		PLC_TX01_Bit_STr_Ack := FALSE;

	end_if;

else

	TP_PB_NoSelTimer(IN:= FALSE);

	OM_PLC_Word1 := INT_TO_WORD(NDC8.OMPLC.ChargeOM);

	OM_PLC_W1_Bit_OM_Cont			:= FALSE;
	OM_PLC_W1_Bit_OM_Finish			:= FALSE;
	OM_PLC_W1_Bit_OM_Cancel			:= FALSE;
	OM_PLC_W1_Bit_OM_Change			:= FALSE;

	NDC8.OMPLC.ChargeOM := WORD_TO_INT(OM_PLC_Word1);

end_if;

PLC_TX_Word3 := 0;

(* I00817 *)
PLC_TX03_Bit_STr_SD_F := Input.SD_Forward;

(* I00818 *)
PLC_TX03_Bit_STr_SD_R := Input.SD_Backward;

(* I00819 *)
PLC_TX03_Bit_STr_Rot_L := Input.SD_Left;

(* I00820 *)
PLC_TX03_Bit_STr_Rot_R := Input.SD_Right;

(* I00821 *)
PLC_TX03_Bit_STr_DD_R := Input.SD_Right;

(* I00822 *)
PLC_TX03_Bit_STr_DD_L := Input.SD_Left;

(* I00823 *)
if g_PlcComLinkUp = TRUE then
	if NDC8.SDIO.DigitalOutput16_Charger = TRUE then
		PLC_TX03_Bit_STr_Charge := TRUE;
	else
		PLC_TX03_Bit_STr_Charge := FALSE;
	end_if;
end_if;

(* I00824 *)
if NDC8.BlockedInfo.BlockedById <> 1 and NDC8.BlockedInfo.BlockedById <> 0 then
	PLC_TX03_Bit_STr_Block := TRUE;
else
	PLC_TX03_Bit_STr_Block := FALSE;
end_if;

(* I00825 *)
if (NDC8.CAN_IO_3.DigitalInput9_AreaF_IN1 = FALSE or NDC8.CAN_IO_3.DigitalInput10_AreaF_IN2 = FALSE) and StopObstacle = TRUE then
	PLC_TX03_Bit_STr_Ir_F := TRUE;
else
	PLC_TX03_Bit_STr_Ir_F := FALSE;
end_if;

(* I00826 *)
if (NDC8.CAN_IO_3.DigitalInput13_AreaR_IN1 = FALSE or NDC8.CAN_IO_3.DigitalInput14_AreaR_IN2 = FALSE) and StopObstacle = TRUE then
	PLC_TX03_Bit_STr_Ir_R := TRUE;
else
	PLC_TX03_Bit_STr_Ir_R := FALSE;
end_if;

(* I00827 *)
	PLC_TX03_Bit_STr_Brake := NDC8.SDIO.DigitalInput5_BTN_BRK;

(* I00828 *)
if NDC8.Autoinsert.StatusID = 1 then
	PLC_TX03_Bit_STr_Search := TRUE;
else
	PLC_TX03_Bit_STr_Search := FALSE;
end_if;

(* I00816 *)
if PLC_TX_Word3 <= 1 then
	PLC_TX03_Bit_STr_Idle := TRUE ;
else
	PLC_TX03_Bit_STr_Idle := FALSE;
end_if;

(* I00832 *)
if NDC8.LayoutPosition.InSystem then
	PLC_TX04_Bit_STr_Ins_dn := TRUE;
else
	PLC_TX04_Bit_STr_Ins_dn := FALSE;
end_if;

(* I00835 *)
(*PLC_TX04_Bit_Cancel_ST := IN_OPCD_Bit_Cmd_EnaEmg;*)
(*InAutoLoad Process*)

(* I00836 *)
RST_Flag := NDC8.SDIO.DigitalInput2_BTN_RST or g_RemoteReset;

RST_R(CLK := RST_Flag);

if RST_R.Q then
	RST_Keep := TRUE;
	RST_Keep_Timer(IN:= FALSE);
end_if;

if RST_Keep = TRUE then
	RST_Keep_Timer(IN:= TRUE, PT := t#1.5s);
end_if;

if RST_Keep_Timer.Q then
	RST_Keep := FALSE;
	RST_Keep_Timer(IN:= FALSE);
end_if;

if PLC_RX_Word20_PLC_ErrD <> 0 then
	PLC_TX04_Bit_Reset_o := RST_Keep;
else
	PLC_TX04_Bit_Reset_o := FALSE;
end_if;

g_AGV_ErrorReset := RST_Keep;

(* I00837 *)
if PLC_TX_Word13_STr_Err <> 0 then
	PLC_TX04_Bit_AgvErr_o := TRUE;
else
	PLC_TX04_Bit_AgvErr_o := FALSE;
end_if;

(* I00838 *)

(*
if StopWord <> 0 then
	PLC_TX04_Bit_AgvErr_o := TRUE;
	PLC_TX_Word13_STr_Err := INT_TO_WORD(DWORD_TO_INT(StopWord));
else
	PLC_TX04_Bit_AgvErr_o := FALSE;
	PLC_TX_Word13_STr_Err := 0;

end_if;
*)

(*I00846*)
if PLC_TX04_Bit_ChkCom_Tx <> PLC_LastHeartBeat then
	PLC_HeartBeatNoChange := false;
else
	PLC_HeartBeatNoChange := true;
end_if;

PLC_LastHeartBeat := PLC_TX04_Bit_ChkCom_Tx;

PLC_HeartBeatTimeout(IN:= PLC_HeartBeatNoChange, PT:= t#10s);

(* D507 *)
PLC_TX_Word7_STr_Vecl := DINT_TO_WORD(NDC8.Vehicle.VehicleID);

(* D508 *)
PLC_TX_Word8_STr_Seg := DINT_TO_WORD(NDC8.LayoutPosition.Segment);

(* D509 *)

if PLC_TX01_Bit_LocalMode then
	if NDC8.LocalOrder.DestPoint <> 0 then
		FinalPnt := NDC8.LocalOrder.DestPoint;
	end_if;
elsif PLC_TX01_Bit_HostMode then
	if NDC8.Automatic.DestPoint <> 0 then
		FinalPnt := NDC8.Automatic.DestPoint;
	end_if;
end_if;

PLC_TX_Word9_STr_Pnt := DINT_TO_WORD(FinalPnt);

(* D510 *)
PLC_TX_Word10_STr_BatV := PLC_RX_Word16_BMS_BatV;

(* D511 *)
PLC_TX_Word11_STr_Temp := PLC_RX_Word17_BMS_BatT;

(* D514 *)
ConvWord := INT_TO_WORD(NDC8.OMPLC.R_BCD3);

WordL := BYTE_TO_INT(ConvByteH);
WordH := BYTE_TO_INT(ConvByteL);
TempInt := WordH * 256 + WordL;
TempWord := INT_TO_WORD(TempInt);

PLC_TX_Word14_STr_BCD3 := TempWord;

(* D515 *)
ConvWord := INT_TO_WORD(NDC8.OMPLC.R_BCD2);

WordL := BYTE_TO_INT(ConvByteH);
WordH := BYTE_TO_INT(ConvByteL);
TempInt := WordH * 256 + WordL;
TempWord := INT_TO_WORD(TempInt);

PLC_TX_Word15_STr_BCD2 := TempWord;

(* D516 *)
ConvWord := INT_TO_WORD(NDC8.OMPLC.R_BCD1);

WordL := BYTE_TO_INT(ConvByteH);
WordH := BYTE_TO_INT(ConvByteL);
TempInt := WordH * 256 + WordL;
TempWord := INT_TO_WORD(TempInt);

PLC_TX_Word16_STr_BCD1 := TempWord;

(*RX Data Proc*)
(*Set Local order mode*)
if PLC_RX03_Bit_STw_Mod_LT and not PLC_RX03_Bit_STw_Mod_NT and not PLC_RX03_Bit_STw_Mod_UT then
	NDC8.Automatic.SetOrderMode := 3;
	OrderMode();
end_if;

LocalManual := NDC8.Mcd.Button3;

LocalManual_R(CLK:= LocalManual);

if LocalManual_R.Q then
	SetToLocal := TRUE;
end_if;

if SetToLocal then
	NDC8.Automatic.SetOrderMode := 3;
	OrderMode();

	if NDC8.Automatic.CurrentOrderMode = 3 then
		SetToLocal := false;
	end_if;
end_if;

if (PLC_RX03_Bit_STw_Mod_LT and PLC_RX03_Bit_STw_Mod_NT) then
	NDC8.Automatic.SetOrderMode := 2;
	OrderMode();
end_if;

if PLC_RX03_Bit_STw_Mod_LT and PLC_RX03_Bit_STw_Mod_UT then
	NDC8.Automatic.SetOrderMode := 3;
	OrderMode();

	if OrderMode.Finished then
		PLC_TX01_Bit_STr_Mod_NT := FALSE;
		PLC_TX01_Bit_STr_Mod_UT := TRUE;
	end_if;
end_if;

(*Set Host order mode*)
if PLC_RX03_Bit_STw_Mod_HT then
	NDC8.Automatic.SetOrderMode := 1;
	OrderMode();
end_if;

(* Set Insert Point *)
if NDC8.LayoutPosition.InSystem = FALSE and PLC_RX_Word11_Ins_Pno <> 0 then

	NDC8.NavInit.Target := Word_To_DINT(PLC_RX_Word11_Ins_Pno);
	NavInit(Method:= 1);
	if NavInit.Finished and NavInit.ErrorCode <> 0 then
		PLC_TX04_Bit_STr_Ins_dn := TRUE;
		PLC_TX04_Bit_STr_Ins_er := FALSE;
	else
		PLC_TX04_Bit_STr_Ins_dn := FALSE;
		PLC_TX04_Bit_STr_Ins_er := TRUE;
	end_if;
end_if;

(* Set Local Order Data*)
STw_NewcmdR(CLK:= PLC_RX03_Bit_STw_Newcmd);

if STw_NewcmdR.Q then
	STw_Newcmd_Flag := TRUE;
end_if;

if STw_Newcmd_Flag then
	NDC8.LocalOrder.DestPoint := Word_To_DINT(PLC_RX_Word12_STw_Pint);
	NDC8.LocalOrder.OpCode := Word_To_DINT(PLC_RX_Word5);
	PLC_TX04_Bit_STr_Cmd_dn := FALSE;

	LocalOrder();
	if LocalOrder.Finished then
		STw_Newcmd_Flag := FALSE;
	end_if;
end_if;

if INPUT.AutoLoadDone then
	PLC_TX04_Bit_STr_Cmd_dn := TRUE;
else
	PLC_TX04_Bit_STr_Cmd_dn := FALSE;
end_if;

if PLC_RX03_Bit_STw_Newcmd = FALSE then
	PLC_TX04_Bit_STr_Cmd_dn := FALSE;
end_if;

(* Battery Voltage*)
if g_PlcComLinkUp = TRUE then
	Input.Display_BatteryLevel := PLC_RX_Word16_BMS_BatV;
else
	Input.Display_BatteryLevel := 0;
end_if;

BMS_BatLowSel := DINT_TO_INT(NDC8.UserDefined.Integer32_51_BattLowSel);

case BMS_BatLowSel of

3:
	BMS_BatLow := PLC_RX15_Bit_BMS_ChgRqH;
2:
	BMS_BatLow := PLC_RX15_Bit_BMS_ChgRqM or PLC_RX15_Bit_BMS_ChgRqH;
1:
	BMS_BatLow := PLC_RX15_Bit_BMS_ChgRqL or PLC_RX15_Bit_BMS_ChgRqM or PLC_RX15_Bit_BMS_ChgRqH;
end_case;

if NDC8.UserDefined.Integer32_50_BattLowVol = 0 or NDC8.UserDefined.Integer32_50_BattLowVol < 0 then
	NDC8.UserDefined.Integer32_50_BattLowVol := 240;
end_if;

if PLC_RX_Word16_BMS_BatV < DINT_TO_WORD(NDC8.UserDefined.Integer32_50_BattLowVol) then
	BatLow := TRUE;
else
	BatLow:= FALSE;
end_if;

if (BMS_BatLow = TRUE or BatLow = TRUE)then
	INPUT.LowBattery := TRUE;
else
	INPUT.LowBattery := FALSE;
end_if;

(* Battery Temperature *)
if g_PlcComLinkUp = TRUE then
	Input.Display_Temperature := PLC_RX_Word17_BMS_BatT;
else
	Input.Display_Temperature := 0;
end_if;

(* Battery Low OT *)
if g_PlcComLinkUp = TRUE then
	g_PowerOffFlag_PLC := PLC_RX04_Bit_STw_LowOT;
end_if;

(*Communication*)

(****************************************************************************)
if ComStart = true then

	if init = true then
		case ComStep of
		0:
		(*StartDelay:=False;
		IF Not StartDelayTOF.Q THEN*)
			ComStep:=1;
		(*END_IF;*)
		(* no delay when PLC <--> CVC700*)
		(****************************************************************************)
		1:

			serial_read();
			msg_index := 0;
			while serial_read.length > 0 do

				(* Copy message to local buffer *)
				for dataindex := 1 to serial_read.length by 1 do
					ix := dataindex + msg_index;
					PLC_message[ix] := serial_read.data[dataindex];
				end_for;
				(* Point for next possible message *)
				msg_index := msg_index + serial_read.length;
				serial_read();
			end_while;

			IF msg_index <> 0 then
				ComStep:=2;
			Else
				ComStep:=0;
			END_IF;

		(****************************************************************************)
		2:
				    (* Parse *)
					tr_cmd := BYTE_TO_DINT(PLC_message[8]);
					tr_len := BYTE_TO_DINT(PLC_message[6]);

					dummy := TRACE_DINT('Cmd', tr_cmd);
					dummy := TRACE_DINT('Len', tr_len);

					(* Copy header *)
					serial_write.data[1] := PLC_message[1];
					serial_write.data[2] := PLC_message[2];
					serial_write.data[3] := PLC_message[3];
					serial_write.data[4] := PLC_message[4];
					serial_write.data[5] := PLC_message[5];		(* Length, will be overwritten *)

					serial_write.data[6] := PLC_message[6]; 	(* Length, will be overwritten *)
					serial_write.data[7] := PLC_message[7]; 	(* Slave adress *)
					serial_write.data[8] := PLC_message[8]; 	(* Cmd *)

					(* Start adress to read *)
					ConvByteH:= PLC_message[9];
					ConvByteL:= PLC_message[10];
					start_adress  := Word_TO_INT(pConvWord) + 1;

					ComStep:=3;

		(****************************************************************************)
		3:

					(*Check Function type *)

					case tr_cmd of
						6:	ComStep:=60;	(* Check if Write single register *)
						16:	ComStep:=160; (* Check if write Multiple register *)
						3:	ComStep:=30;	(*Check if Read register *)
					Else
						ComStep:=999; 	(*Send Echo *)
					end_case;

		(****************************************************************************)
		30:
						(*Read register *)
						(* Number of words *)
						(* serial_read.data[11]; *)
						(*CVC700 -> PLC HandShake Data*)
						PLC_Communication_ModBus_ValueWord [1] := PLC_TX_Word1;
						PLC_Communication_ModBus_ValueWord [2] := PLC_TX_Word2;
						PLC_Communication_ModBus_ValueWord [3] := PLC_TX_Word3;
						PLC_Communication_ModBus_ValueWord [4] := PLC_TX_Word4;
						PLC_Communication_ModBus_ValueWord [5] := PLC_TX_Word5;
						PLC_Communication_ModBus_ValueWord [6] := PLC_TX_Word6;
						PLC_Communication_ModBus_ValueWord [7] := PLC_TX_Word7_STr_Vecl;
						PLC_Communication_ModBus_ValueWord [8] := PLC_TX_Word8_STr_Seg;
						PLC_Communication_ModBus_ValueWord [9] := PLC_TX_Word9_STr_Pnt;
						PLC_Communication_ModBus_ValueWord [10] := PLC_TX_Word10_STr_BatV;
						PLC_Communication_ModBus_ValueWord [11] := PLC_TX_Word11_STr_Temp;
						PLC_Communication_ModBus_ValueWord [12] := PLC_TX_Word12_STr_BatD;
						PLC_Communication_ModBus_ValueWord [13] := PLC_TX_Word13_STr_Err;
						PLC_Communication_ModBus_ValueWord [14] := PLC_TX_Word14_STr_BCD3;
						PLC_Communication_ModBus_ValueWord [15] := PLC_TX_Word15_STr_BCD2;
						PLC_Communication_ModBus_ValueWord [16] := PLC_TX_Word16_STr_BCD1;
						num_words := BYTE_TO_DINT(PLC_message[12]);

						IF num_words >21 THEN
						   		num_words:=21;
							END_IF;

							(*Y:=start_adress;*)
							Y := 1;
							(*Z:=10;*)
							Z:= 1; (* Send first 9*)
							Serial_write.data[1] := DINT_TO_BYTE(255);
							Serial_write.data[9] := DINT_TO_BYTE(32);
							serial_write.data[6] := DINT_TO_BYTE(35); (* lp *)
				        	serial_write.length := 9;
							serial_write();
							serial_write.length := 0;
							serial_write(); (*send*)
							Counter := 16;	(*send the rest words*)
							WHILE Counter > 0 do
								lenght_send := MIN(16,Counter); (*Can max send 32bytes in 1 serial_write so need to make sure for-loop gets correct number of itterations*)
								For Index:=1 to 16 BY 1 DO
									pConvWord:=PLC_Communication_ModBus_ValueWord [Y];
									serial_write.data[Z]:=pConvByteH;
									Z:=Z+1;
									serial_write.data[Z]:=pConvByteL;
									Z:=Z+1;
									Y:=Y+1;
								END_FOR;
								serial_write.length := DINT_TO_INT(32); (*Will be max 32 bytes*)
								serial_write();
								Counter := Counter - lenght_send; (*Count down for while loop*)
							END_WHILE;
							serial_write.length := 0; (*Using SendBuffer =1 length needs to be set to 0 for it to be sent*)
							serial_write(); (*send*)

							ComStep:=10001;

			(****************************************************************************)
		60:
						(* Write single register *)
						(* single write *)
						(* Number of words *)
						(* serial_read.data[11]; *)
						num_words := BYTE_TO_DINT(PLC_message[12]);
						Y:=start_adress;
						pConvByteH:=PLC_message[11];
					    pConvByteL:=PLC_message[12];
						PLC_Communication_ModBus_ValueWord [Y]:=pConvWord;

						ComStep:=999;
		(****************************************************************************)
		160:
						(* Multiple write *)
						num_words:=Byte_TO_DInt(PLC_message[12]);
						(* Check if message lenght outside the Buffer, if so do what ??? *)
						IF num_words > 25 THEN
						   num_words:=25;
						END_IF;
						Y:=17;
						X:=14;  (*13 = 後面要寫入的資料位元組數，0x08=十進位制8，寫8個位元組 , 忽略*)
						End:= Byte_TO_Int(PLC_message[12]);

						For Index:=1 to num_words BY 1 DO
							pConvByteH:=PLC_message[X];
							X:=X+1;
							pConvByteL:=PLC_message[X];
							ModBus_ValueWord [Y]:=pConvWord;
							X:=X+1;
							Y:=Y+1;
						END_FOR;
						(*Set Into Memory *)
						PLC_RX_Word1 := PLC_Communication_ModBus_ValueWord [17];
						PLC_RX_Word2 := PLC_Communication_ModBus_ValueWord [18];
						PLC_RX_Word3 := PLC_Communication_ModBus_ValueWord [19];
						PLC_RX_Word4 := PLC_Communication_ModBus_ValueWord [20];
						PLC_RX_Word5 := PLC_Communication_ModBus_ValueWord [21];
						PLC_RX_Word6 := PLC_Communication_ModBus_ValueWord [22];
						PLC_RX_Word7_STw_BCD3 := PLC_Communication_ModBus_ValueWord [23];
						PLC_RX_Word8_STw_BCD2 := PLC_Communication_ModBus_ValueWord [24];
						PLC_RX_Word9_STw_BCD1 := PLC_Communication_ModBus_ValueWord [25];
						PLC_RX_Word10_STw_ILEr := PLC_Communication_ModBus_ValueWord [26];
						PLC_RX_Word11_Ins_Pno := PLC_Communication_ModBus_ValueWord [27];
						PLC_RX_Word12_STw_Pint := PLC_Communication_ModBus_ValueWord [28];
						PLC_RX_Word13_Ins_Ano := PLC_Communication_ModBus_ValueWord [29];
						PLC_RX_Word14_BMS_2 := PLC_Communication_ModBus_ValueWord [30];
						PLC_RX_Word15_BMS_3 := PLC_Communication_ModBus_ValueWord [31];
						PLC_RX_Word16_BMS_BatV := PLC_Communication_ModBus_ValueWord [32];
						PLC_RX_Word17_BMS_BatT := PLC_Communication_ModBus_ValueWord [33];
						PLC_RX_Word18_BMS_BatC := PLC_Communication_ModBus_ValueWord [34];
						PLC_RX_Word19_BMS_BatA := PLC_Communication_ModBus_ValueWord [35];
						PLC_RX_Word20_PLC_ErrD := PLC_Communication_ModBus_ValueWord [36];
						PLC_RX_Word21_BMS_Main := PLC_Communication_ModBus_ValueWord [37];
						PLC_RX_Word22_BMS_Chan := PLC_Communication_ModBus_ValueWord [38];
						PLC_RX_Word23_BMS_ID4L := PLC_Communication_ModBus_ValueWord [39];
						PLC_RX_Word24_BMS_ID4H := PLC_Communication_ModBus_ValueWord [40];
						PLC_RX_Word25 := PLC_Communication_ModBus_ValueWord [41];

						ComStep:=999;
		(****************************************************************************)
		999:

						(*Send Echo *)
							Serial_write.data[9] := PLC_message[9];
							serial_write.data[10] := PLC_message[10];
							serial_write.data[11] := PLC_message[11];
							serial_write.data[12] := PLC_message[12];

							length :=6;
							tx_length := DINT_TO_BYTE(length);
					        serial_write.data[6] := tx_length; (* lp *)
							ComStep:=10000;

		(****************************************************************************)
		10000:

					(*Send Data *)

					serial_write.length := BYTE_TO_INT(tx_header_length) + BYTE_TO_INT(tx_length);
					serial_write();

					serial_write.length := 0;
					serial_write();

					IF serial_write.sent<>0 or serial_write.error<>0 Then
						ComStep:=0;
						DebugCounter := DebugCounter + 1;
					End_IF;
		10001:
					IF serial_write.sent<>0 or serial_write.error<>0 Then
						ComStep:=0;
						DebugCounter := DebugCounter + 1;
					End_IF;
		end_case;

	(*CVC700 -> PLC HandShake Data*)
	(*PLC_Communication_ModBus_ValueWord [1] := PLC_TX_Word1;
	PLC_Communication_ModBus_ValueWord [2] := PLC_TX_Word2;
	PLC_Communication_ModBus_ValueWord [3] := PLC_TX_Word3;
	PLC_Communication_ModBus_ValueWord [4] := PLC_TX_Word4;
	PLC_Communication_ModBus_ValueWord [5] := PLC_TX_Word5;
	PLC_Communication_ModBus_ValueWord [6] := PLC_TX_Word6;
	PLC_Communication_ModBus_ValueWord [7] := PLC_TX_Word7_STr_Vecl;
	PLC_Communication_ModBus_ValueWord [8] := PLC_TX_Word8_STr_Seg;
	PLC_Communication_ModBus_ValueWord [9] := PLC_TX_Word9_STr_Pnt;
	PLC_Communication_ModBus_ValueWord [10] := PLC_TX_Word10_STr_BatV;
	PLC_Communication_ModBus_ValueWord [11] := PLC_TX_Word11_STr_Temp;
	PLC_Communication_ModBus_ValueWord [12] := PLC_TX_Word12_STr_BatD;
	PLC_Communication_ModBus_ValueWord [13] := PLC_TX_Word13_STr_Err;
	PLC_Communication_ModBus_ValueWord [14] := PLC_TX_Word14_STr_BCD3;
	PLC_Communication_ModBus_ValueWord [15] := PLC_TX_Word15_STr_BCD2;
	PLC_Communication_ModBus_ValueWord [16] := PLC_TX_Word16_STr_BCD1;
	*)

	(*PLC -> CVC700 HandShake Data*)
	(*PLC_RX_Word1 := PLC_Communication_ModBus_ValueWord [17];
	PLC_RX_Word2 := PLC_Communication_ModBus_ValueWord [18];
	PLC_RX_Word3 := PLC_Communication_ModBus_ValueWord [19];
	PLC_RX_Word4 := PLC_Communication_ModBus_ValueWord [20];
	PLC_RX_Word5 := PLC_Communication_ModBus_ValueWord [21];
	PLC_RX_Word6 := PLC_Communication_ModBus_ValueWord [22];
	PLC_RX_Word7_STw_BCD3 := PLC_Communication_ModBus_ValueWord [23];
	PLC_RX_Word8_STw_BCD2 := PLC_Communication_ModBus_ValueWord [24];
	PLC_RX_Word9_STw_BCD1 := PLC_Communication_ModBus_ValueWord [25];
	PLC_RX_Word10_STw_ILEr := PLC_Communication_ModBus_ValueWord [26];
	PLC_RX_Word11_Ins_Pno := PLC_Communication_ModBus_ValueWord [27];
	PLC_RX_Word12_STw_Pint := PLC_Communication_ModBus_ValueWord [28];
	PLC_RX_Word13_Ins_Ano := PLC_Communication_ModBus_ValueWord [29];
	PLC_RX_Word14_BMS_2 := PLC_Communication_ModBus_ValueWord [30];
	PLC_RX_Word15_BMS_3 := PLC_Communication_ModBus_ValueWord [31];
	PLC_RX_Word16_BMS_BatV := PLC_Communication_ModBus_ValueWord [32];
	PLC_RX_Word17_BMS_BatT := PLC_Communication_ModBus_ValueWord [33];
	PLC_RX_Word18_BMS_BatC := PLC_Communication_ModBus_ValueWord [34];
	PLC_RX_Word19_BMS_BatA := PLC_Communication_ModBus_ValueWord [35];
	PLC_RX_Word20_PLC_ErrD := PLC_Communication_ModBus_ValueWord [36];
	PLC_RX_Word21_BMS_Main := PLC_Communication_ModBus_ValueWord [37];
	PLC_RX_Word22_BMS_Chan := PLC_Communication_ModBus_ValueWord [38];
	PLC_RX_Word23_BMS_ID4L := PLC_Communication_ModBus_ValueWord [39];
	PLC_RX_Word24_BMS_ID4H := PLC_Communication_ModBus_ValueWord [40];
	PLC_RX_Word25 := PLC_Communication_ModBus_ValueWord [41];
	*)
	end_if;

end_if;

END_FUNCTION_BLOCK
